// TIA Portal V20 export
// export: Created 2025-12-01T14:57:46.9707889Z, ExportSetting None, DisplayName Totally Integrated Automation Portal, DisplayVersion V20 Update 3, DisplayName TIA Portal Openness, DisplayVersion V20 Update 3, DisplayName TIA Portal Version Control Interface, DisplayVersion V20 Update 3, DisplayName STEP 7 Professional, DisplayVersion V20 Update 3, DisplayName STEP 7 Safety, DisplayVersion V20 Update 2, DisplayName WinCC Basic/Comfort/Advanced, DisplayVersion V20 Update 3, DisplayName WinCC Professional, DisplayVersion V20 Update 3, DisplayName WinCC Unified, DisplayVersion V20 Update 3
DATA_BLOCK "DB214_CNT_Mens_SCR"   // DB214
{ S7_Optimized_Access := 'FALSE' }
AUTHOR : ROUTER
NAME : 20130623
VERSION : 3.1
// stored: AutoNumber false
   VAR RETAIN
      RedScanners : Array[1..5] of Struct
         CNT_NODO_PROF_SCR : Array[0..254] of Byte;   // No puedo acceder directamente a cargar una dirección PA de los scanners.
      END_STRUCT;
   END_VAR
BEGIN
END_DATA_BLOCK
